Staubli VAL3: stop.pgx

program stop()
begin
  disablePower()
  resetMotion()
  $fileClose(0)
  $fileClose(1)
  $fileClose(2)
  $fileClose(3)
  $fileClose(4)
  $fileClose(5)
  $fileClose(6)
  $fileClose(7)
  $fileClose(8)
   libSave()


end
